(* CODESYS project Lift Demo 1.project

Project tree, tasks and I/O mapping:
  Device : CODESYS Control Win V3, 3S - Smart Software Solutions GmbH, version 3.5.16.70
    application Application
      libraries: Standard, * (System)
      task MainTask (cyclic, interval t#20ms, priority 1) calls Simulatie, Demo1
      visualisation Visualization
  Lift Besturing/
    program DeurBesturing [ST]
  global variables GVL
  image pool ImagePool
  5ce3da45-db07-42e7-a21c-a00fff4ed8f6|C:\Users\Gerard\Desktop\MensenInLift.PNG
  5ce3da45-db07-42e7-a21c-a00fff4ed8f6|C:\Users\Gerard\Desktop\LiftDeur.PNG
  5ce3da45-db07-42e7-a21c-a00fff4ed8f6|C:\Users\Gerard\Desktop\Liftaandrijving.PNG
  5ce3da45-db07-42e7-a21c-a00fff4ed8f6|C:\Users\Gerard\Desktop\LiftDeurAandrijving.PNG
  Lift Simualtie/
    program Simulatie [ST]
  text list GlobalTextList
  Demo/
    program Demo1 [ST]
    program Demo2 [ST]
    program Demo3 [ST]
*)

// GVL
VAR_GLOBAL
	Ix_BovenOproepKooi					: BOOL;
	Ix_BenedenOproepKooi				: BOOL;
	Ix_KooiGaNaarBoven					: BOOL;
	Ix_KooiGaNaarBeneden				: BOOL;
	Ix_KooiBoven						: BOOL;
	Ix_KooiBeneden						: BOOL;
	Qx_AandrijvingOmhoog				: BOOL;
	Qx_AandrijvingOmlaag				: BOOL;
	
	
	Ix_BenedenDeurOpen					: BOOL;
	Ix_BenedenDeurGesloten				: BOOL;
	Qx_BenedenDeurAandrijvingOpen		: BOOL;
	Qx_BenedenDeurAandrijvingSluiten	: BOOL;
	
	Ix_BovenDeurOpen					: BOOL;
	Ix_BovenDeurGesloten				: BOOL;
	Qx_BovenDeurAandrijvingOpen			: BOOL;
	Qx_BovenDeurAandrijvingSluiten		: BOOL;
	
	Ix_TestKnop1						: BOOL;
	Ix_TestKnop2						: BOOL;
	Qx_TestLamp1						: BOOL;
	Qx_TestLamp2						: BOOL;
	
END_VAR

// Lift Simualtie/Simulatie
// Programma		: Simulatie
// Project			: Lift
// Doel				: Simulatie functies voor de lift
// Auteur			: Gerard Harkema
// Versie			: 1.0
// Datum			: 15 oktober 2015

PROGRAM Simulatie
VAR
	FB_PulsgeverTimer					: TON;
	Mw_PulsgeverTimerPT					: TIME := T#10MS;
	Mx_PulsLiftAandrijving				: BOOL;
	Mx_Pulsgever						: BOOL;
	Mw_PelsgeverTimerET					: TIME;
	FB_SnelheidLift						: CTU;
	Mw_SnelheidLiftPV					: WORD := 4;
	Mw_SnelheidLiftCV					: WORD;

	Mw_PositieLiftInv					: INT := 0;
	Mw_PositieLift						: INT := 0;
	Mw_LiftBenedenCountValue			: INT := 250;

	Mw_BenedenPositieDeur				: INT := 0;
	Mw_BenedenPositieDeurCountValue		: INT := 100;

	Mw_BovenPositieDeur					: INT := 40;
	Mw_BovenPositieDeurCountValue		: INT := 100;

END_VAR

// Puls gever voor de bewegings simualties

FB_PulsgeverTimer(IN:= (NOT Mx_Pulsgever),PT:= Mw_PulsgeverTimerPT ,Q => Mx_Pulsgever, ET => Mw_PelsgeverTimerET);

//*********************************************
//                 Lift
//*********************************************

// Snelheid lift
FB_SnelheidLift(CU := Mx_Pulsgever, RESET := Mx_PulsLiftAandrijving, PV := Mw_SnelheidLiftPV, Q => Mx_PulsLiftAandrijving, CV => Mw_SnelheidLiftCV);

// Detectie lift is boven
IF (Mw_PositieLiftInv >= Mw_LiftBenedenCountValue) THEN
	GVL.Ix_KooiBoven := TRUE;
ELSE
	GVL.Ix_KooiBoven := FALSE;	
END_IF
  

// Detectie lift is beneden
IF(Mw_PositieLiftInv <= 0) THEN
	GVL.Ix_KooiBeneden := TRUE;
ELSE
	GVL.Ix_KooiBeneden := FALSE;	
END_IF


// Reizen lift omhoog
IF(GVL.Qx_AandrijvingOmhoog AND Mx_PulsLiftAandrijving AND (NOT GVL.Ix_KooiBoven)) THEN
	Mw_PositieLiftInv := Mw_PositieLiftInv + 5;
END_IF

// Reizen lift omlaag
IF(GVL.Qx_AandrijvingOmlaag AND Mx_PulsLiftAandrijving AND (NOT GVL.Ix_KooiBeneden)) THEN
	Mw_PositieLiftInv := Mw_PositieLiftInv - 5;
END_IF

Mw_PositieLift := Mw_LiftBenedenCountValue - Mw_PositieLiftInv;


// Inactief maken oproepknoppen
IF GVL.Ix_KooiBoven THEN
 Ix_BovenOproepKooi := FALSE;
END_IF

IF GVL.Ix_KooiBoven THEN
 Ix_KooiGaNaarBoven := FALSE;
END_IF


IF GVL.Ix_KooiBeneden THEN
 Ix_BenedenOproepKooi := FALSE;
END_IF

IF GVL.Ix_KooiBeneden THEN
 Ix_KooiGaNaarBeneden := FALSE;
END_IF
 

//*********************************************
//                 Benedendeur
//*********************************************

// Detectie Benedendeur is open
IF (Mw_BenedenPositieDeur >= Mw_BenedenPositieDeurCountValue) THEN
	GVL.Ix_BenedenDeurOpen := TRUE;
ELSE
	GVL.Ix_BenedenDeurOpen := FALSE;	
END_IF
  

// Detectie Benedendeur is gesloten
IF(Mw_BenedenPositieDeur <= 0) THEN
	GVL.Ix_BenedenDeurGesloten := TRUE;
ELSE
	GVL.Ix_BenedenDeurGesloten := FALSE;	
END_IF


// Benedendeur openen
IF(GVL.Qx_BenedenDeurAandrijvingOpen AND Mx_PulsLiftAandrijving AND (NOT GVL.Ix_BenedenDeurOpen)) THEN
	Mw_BenedenPositieDeur := Mw_BenedenPositieDeur + 5;
END_IF

// Benedendeur sluiten
IF(GVL.Qx_BenedenDeurAandrijvingSluiten AND Mx_PulsLiftAandrijving AND (NOT GVL.Ix_BenedenDeurGesloten)) THEN
	Mw_BenedenPositieDeur := Mw_BenedenPositieDeur - 5;
END_IF

//*********************************************
//                 Bovendeur
//*********************************************

// Detectie bovendeur is open
IF (Mw_BovenPositieDeur >= Mw_BovenPositieDeurCountValue) THEN
	GVL.Ix_BovenDeurOpen := TRUE;
ELSE
	GVL.Ix_BovenDeurOpen := FALSE;	
END_IF
  

// Detectie bovendeur is gesloten
IF(Mw_BovenPositieDeur <= 0) THEN
	GVL.Ix_BovenDeurGesloten := TRUE;
ELSE
	GVL.Ix_BovenDeurGesloten := FALSE;	
END_IF


// Bovendeur openen
IF(GVL.Qx_BovenDeurAandrijvingOpen AND Mx_PulsLiftAandrijving AND (NOT GVL.Ix_BovenDeurOpen)) THEN
	Mw_BovenPositieDeur := Mw_BovenPositieDeur + 5;
END_IF

// Bovendeur sluiten
IF(GVL.Qx_BovenDeurAandrijvingSluiten AND Mx_PulsLiftAandrijving AND (NOT GVL.Ix_BovenDeurGesloten)) THEN
	Mw_BovenPositieDeur := Mw_BovenPositieDeur - 5;
END_IF

END_PROGRAM

// Demo/Demo1
PROGRAM Demo1
VAR
	// Variabelen lijst
	xGaSluiten		: BOOL := FALSE;
	xGaOpen			: BOOL := FALSE;
	xOpen			: BOOL;
	xDicht			: BOOL;
	xFirstRun		: BOOL := TRUE;
END_VAR

// Programma
IF xFirstRun THEN
	Qx_BovenDeurAandrijvingSluiten := TRUE;
	xFirstRun := FALSE;
END_IF

xGaSluiten := Ix_TestKnop1;
xGaOpen := Ix_TestKnop2;

xOpen := Ix_BovenDeurOpen;
xDicht := Ix_BovenDeurGesloten;

IF Ix_BovenDeurOpen AND xGaSluiten THEN
	Ix_TestKnop1 := FALSE;
	Qx_BovenDeurAandrijvingSluiten := TRUE;
END_IF;

IF Ix_BovenDeurGesloten THEN
	Qx_BovenDeurAandrijvingSluiten := FALSE;
END_IF;

IF Ix_BovenDeurGesloten AND xGaOpen THEN
	Ix_TestKnop2 := FALSE;
	Qx_BovenDeurAandrijvingOpen := TRUE;
END_IF;

IF Ix_BovenDeurOpen THEN
	Qx_BovenDeurAandrijvingOpen := FALSE;
END_IF;

Qx_TestLamp1 := xOpen;
Qx_TestLamp2 := xDicht;

END_PROGRAM

// Demo/Demo2
PROGRAM Demo2
VAR
	// Variabelen lijst
	xGaSluiten		: BOOL := FALSE;
	xGaOpen			: BOOL := FALSE;
	xOpen			: BOOL;
	xDicht			: BOOL;
	xFirstRun		: BOOL := TRUE;
	
	fbOpenDelay		: TON;
	tOpenDelayPT	: TIME := T#5S;
	tOpenDelayET	: TIME;
	xGaOpenDelay	: BOOL;
	
END_VAR

// Programma
IF xFirstRun THEN
	Qx_BovenDeurAandrijvingSluiten := TRUE;
	xFirstRun := FALSE;
END_IF

xGaSluiten := Ix_TestKnop1;
xGaOpen := Ix_TestKnop2;


xOpen := Ix_BovenDeurOpen;
xDicht := Ix_BovenDeurGesloten;

fbOpenDelay(IN:= Ix_BovenDeurGesloten AND xGaOpen,PT:= tOpenDelayPT ,Q => xGaOpenDelay, ET => tOpenDelayET);


IF Ix_BovenDeurOpen AND xGaSluiten THEN
	Ix_TestKnop1 := FALSE;
	Qx_BovenDeurAandrijvingSluiten := TRUE;
END_IF;

IF Ix_BovenDeurGesloten THEN
	Qx_BovenDeurAandrijvingSluiten := FALSE;
END_IF;

IF xGaOpenDelay THEN
	Ix_TestKnop2 := FALSE;
	Qx_BovenDeurAandrijvingOpen := TRUE;
END_IF;

IF Ix_BovenDeurOpen THEN
	Qx_BovenDeurAandrijvingOpen := FALSE;
END_IF;

Qx_TestLamp1 := xOpen;
Qx_TestLamp2 := xDicht;

END_PROGRAM

// Demo/Demo3
PROGRAM Demo3
VAR
	// Variabelen lijst
	xGaSluiten		: BOOL := FALSE;
	xGaOpen			: BOOL := FALSE;
	xOpen			: BOOL;
	xDicht			: BOOL;
	xFirstRun		: BOOL := TRUE;
	xBovenDeurGeslotenOld: BOOL := FALSE;;
	
	uiTeller		: UINT := 0;
	uiTellerPV		: UINT := 5;
END_VAR

// Programma
IF xFirstRun THEN
	Qx_BovenDeurAandrijvingSluiten := TRUE;
	xFirstRun := FALSE;
END_IF

xGaSluiten := Ix_TestKnop1;
xGaOpen := Ix_TestKnop2;


xOpen := Ix_BovenDeurOpen;
xDicht := Ix_BovenDeurGesloten;

IF (uiTeller = 0) AND Ix_BovenDeurGesloten AND xGaOpen THEN
	uiTeller := uiTellerPV;
	Ix_TestKnop2 := FALSE;
END_IF

IF (uiTeller > 0) AND Ix_BovenDeurGesloten THEN
	Qx_BovenDeurAandrijvingOpen := TRUE;
END_IF


// Flank detectie op gesloten deur
IF (NOT Ix_BovenDeurGesloten) AND xBovenDeurGeslotenOld THEN
	uiTeller := uiTeller - 1;
END_IF
xBovenDeurGeslotenOld := Ix_BovenDeurGesloten;

IF Ix_BovenDeurOpen THEN
	Qx_BovenDeurAandrijvingSluiten := TRUE;
END_IF;

IF Ix_BovenDeurGesloten THEN
	Qx_BovenDeurAandrijvingSluiten := FALSE;
END_IF;

IF Ix_BovenDeurOpen THEN
	Qx_BovenDeurAandrijvingOpen := FALSE;
END_IF;


Qx_TestLamp1 := xOpen;
Qx_TestLamp2 := xDicht;

END_PROGRAM

// Lift Besturing/DeurBesturing
PROGRAM DeurBesturing
VAR
	xGaSluit: BOOL := FALSE;
	xGaOpen: BOOL := FALSE;
	xOpen: BOOL;
	xDicht: BOOL;
END_VAR

IF xGaSluit AND Ix_BovenDeurOpen THEN
	Qx_BovenDeurAandrijvingSluiten := TRUE;
END_IF

IF Ix_BovenDeurGesloten THEN
	Qx_BovenDeurAandrijvingSluiten := FALSE;
END_IF

IF xGaOpen AND Ix_BovenDeurGesloten THEN
	Qx_BovenDeurAandrijvingOpen := TRUE;
END_IF

IF Ix_BovenDeurOpen THEN
	Qx_BovenDeurAandrijvingOpen := FALSE;	
END_IF

xOpen := Ix_BovenDeurOpen;
xDicht := Ix_BovenDeurGesloten;

xGaSluit := Ix_TestKnop1;
xGaOpen := Ix_TestKnop2;

Qx_TestLamp1 := xOpen;
Qx_TestLamp2 := xDicht;

END_PROGRAM

// Device/Application/Visualization
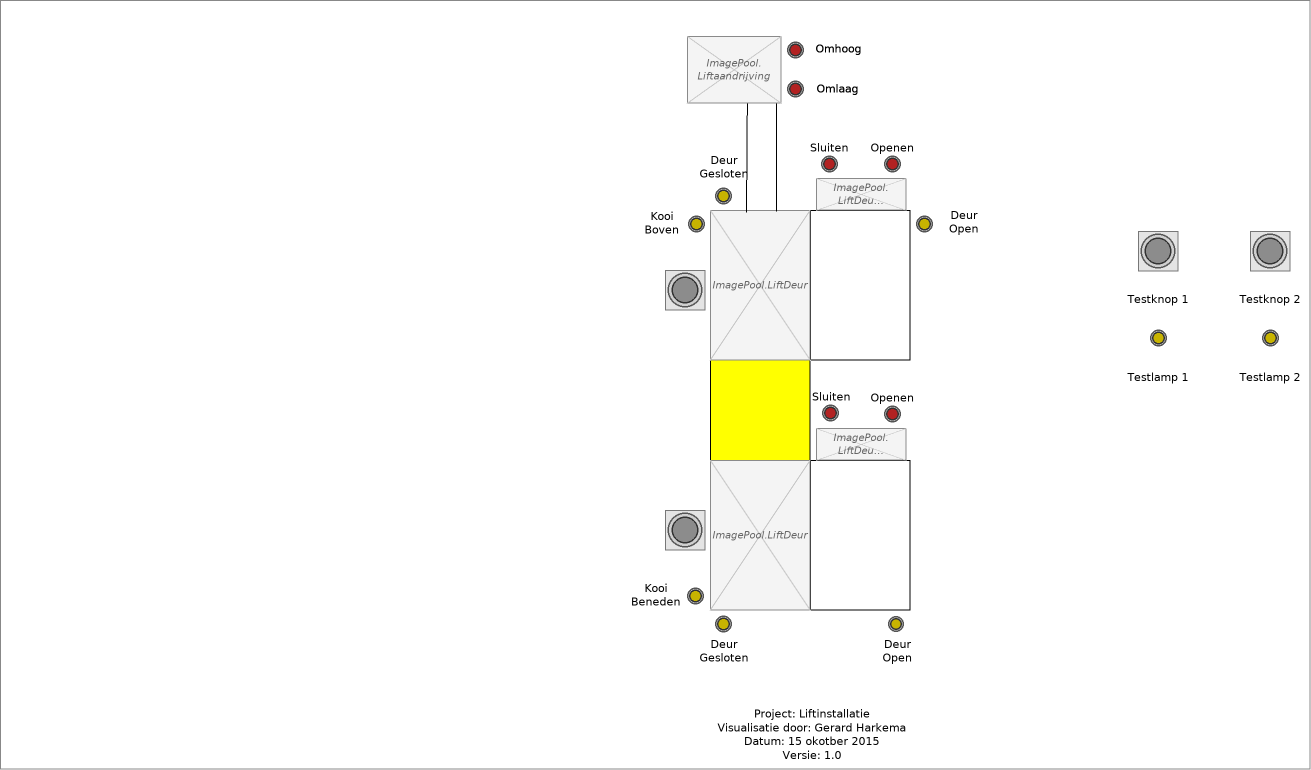
VISUALIZATION Visualization  // 1311x770
    Rectangle (810,460 100x150)
    Rectangle (810,210 100x150)
    Rectangle (710,210 100x400)
    PushSwitch (665,270 40x40), tooltip "Oproep Boven", variable: Ix_BovenOproepKooi, behaviour: TOGGLE, style: Switch-PushSwitch-Gray
    PushSwitch (665,510 40x40), tooltip "Oproep Beneden", variable: Ix_BenedenOproepKooi, behaviour: TOGGLE, style: Switch-PushSwitch-Gray
    Group (710,210 100x150)
        p2738717112: Simulatie.Mw_PositieLift
        Rectangle (0,0 100x150)
        Image (6,0 89x150), image: ImagePool.MensenInLift
        PushSwitch (5,100 30x30), tooltip "Ga naar beneden", variable: Ix_KooiGaNaarBeneden, behaviour: TOGGLE, style: Switch-PushSwitch-Gray
        PushSwitch (5,60 30x30), tooltip "Ga naar Boven", variable: Ix_KooiGaNaarBoven, behaviour: TOGGLE, style: Switch-PushSwitch-Gray
    Rectangle (710,210 100x150)
    Image (716,210 89x150), image: ImagePool.MensenInLift
    PushSwitch (715,310 30x30), tooltip "Ga naar beneden", variable: Ix_KooiGaNaarBeneden, behaviour: TOGGLE, style: Switch-PushSwitch-Gray
    PushSwitch (715,270 30x30), tooltip "Ga naar Boven", variable: Ix_KooiGaNaarBoven, behaviour: TOGGLE, style: Switch-PushSwitch-Gray
    Lamp1 (714,186 19x20), variable: Ix_BovenDeurGesloten, style: Lamp-Lamp1-Yellow
    Lamp1 (915,214 19x20), variable: Ix_BovenDeurOpen, style: Lamp-Lamp1-Yellow
    Lamp1 (687,214 19x20), variable: Ix_KooiBoven, style: Lamp-Lamp1-Yellow
    Lamp1 (686,586 19x20), variable: Ix_KooiBeneden, style: Lamp-Lamp1-Yellow
    Lamp1 (714,614 19x20), variable: Ix_BenedenDeurGesloten, style: Lamp-Lamp1-Yellow
    Lamp1 (887,614 18x20), variable: Ix_BenedenDeurOpen, style: Lamp-Lamp1-Yellow
    Label (682,152 84x30), "Deur Gesloten"
    Label (937,207 54x30), "Deur Open"
    Label (640,208 44x30), "Kooi Boven"
    Label (629,580 54x30), "Kooi Beneden"
    Label (693,636 62x30), "Deur Gesloten"
    Label (875,636 45x30), "Deur Open"
    Group (710,210 100x150)
        p3560616238: Simulatie.Mw_BovenPositieDeur
        Rectangle (0,0 100x150)
        Image (0,0 100x150), image: ImagePool.LiftDeur
    Group (710,460 100x150)
        p3560616238: Simulatie.Mw_BenedenPositieDeur
        Rectangle (0,0 100x150)
        Image (0,0 100x150), image: ImagePool.LiftDeur
    Line (747,83) (746,212)
    Line (776,82) (776,211)
    Group (687,34 182x70)
        Image (0,2 94x67), image: ImagePool.Liftaandrijving
        Lamp1 (99,6 19x20), variable: Qx_AandrijvingOmhoog, style: Lamp-Lamp1-Red
        Lamp1 (99,45 19x20), variable: Qx_AandrijvingOmlaag, style: Lamp-Lamp1-Red
        Label (121,0 61x30), "Omhoog"
        Label (123,40 55x30), "Omlaag"
    Image (687,36 94x67), image: ImagePool.Liftaandrijving
    Lamp1 (786,40 19x20), variable: Qx_AandrijvingOmhoog, style: Lamp-Lamp1-Red
    Lamp1 (786,79 19x20), variable: Qx_AandrijvingOmlaag, style: Lamp-Lamp1-Red
    Label (808,34 61x30), "Omhoog"
    Label (810,74 55x30), "Omlaag"
    Group (816,154 90x56)
        Image (0,24 90x32), image: ImagePool.LiftDeurAandrijving
        Lamp1 (4,0 19x20), variable: Qx_BovenDeurAandrijvingSluiten, style: Lamp-Lamp1-Red
        Lamp1 (67,0 19x20), variable: Qx_BovenDeurAandrijvingOpen, style: Lamp-Lamp1-Red
    Image (816,178 90x32), image: ImagePool.LiftDeurAandrijving
    Lamp1 (820,154 19x20), variable: Qx_BovenDeurAandrijvingSluiten, style: Lamp-Lamp1-Red
    Lamp1 (883,154 19x20), variable: Qx_BovenDeurAandrijvingOpen, style: Lamp-Lamp1-Red
    Group (816,403 90x57)
        Image (0,25 90x32), image: ImagePool.LiftDeurAandrijving
        Lamp1 (5,0 19x20), variable: Qx_BenedenDeurAandrijvingSluiten, style: Lamp-Lamp1-Red
        Lamp1 (67,1 19x20), variable: Qx_BenedenDeurAandrijvingOpen, style: Lamp-Lamp1-Red
    Image (816,428 90x32), image: ImagePool.LiftDeurAandrijving
    Lamp1 (821,403 19x20), variable: Qx_BenedenDeurAandrijvingSluiten, style: Lamp-Lamp1-Red
    Lamp1 (883,404 19x20), variable: Qx_BenedenDeurAandrijvingOpen, style: Lamp-Lamp1-Red
    Label (812,382 39x30), "Sluiten"
    Label (810,133 39x30), "Sluiten"
    Label (867,383 51x30), "Openen"
    Label (867,133 51x30), "Openen"
    Label (712,701 200x67), "Project: Liftinstallatie Visualisatie door: Gerard Harkema Datum: 15 okotber 2015 Versie: 1.0"
    PushSwitch (1138,231 40x40), tooltip "Testknop 1", variable: Ix_TestKnop1, behaviour: TOGGLE, style: Switch-PushSwitch-Gray
    Label (1119,286 78x27), "Testknop 1"
    PushSwitch (1250,231 40x40), tooltip "Testknop 2", variable: Ix_TestKnop2, behaviour: TOGGLE, style: Switch-PushSwitch-Gray
    Label (1231,286 78x27), "Testknop 2"
    Lamp1 (1149,328 19x20), tooltip "Testlamp 1", variable: Qx_TestLamp1, style: Lamp-Lamp1-Yellow
    Lamp1 (1261,328 19x20), tooltip "Testlamp 2", variable: Qx_TestLamp2, style: Lamp-Lamp1-Yellow
    Label (1119,364 78x27), "Testlamp 1"
    Label (1231,364 78x27), "Testlamp 2"
END_VISUALIZATION
